(* IEC 61131-3 sources: Building-Automation/Wastewater Treatment Plant/plc, 7 files *)

(* ---- global_vars.st ---- *)
(* Wastewater Treatment Plant - Global Variables *)
VAR_GLOBAL
    (* Digital Inputs *)
    INTAKE_FLOW AT %I0.0 : BOOL;              (* Intake flow switch *)
    OUTFLOW_SENSOR AT %I0.1 : BOOL;           (* Treated water flow *)
    TANK_HIGH_LEVEL AT %I0.2 : BOOL;          (* High level switch *)
    EMERGENCY_STOP AT %I0.3 : BOOL;           (* Emergency stop *)
    SCREEN_CLOG AT %I0.4 : BOOL;              (* Screen clog detection *)
    AERATION_RUNNING AT %I0.5 : BOOL;         (* Aeration status *)
    PUMP_P101_RUNNING AT %I0.6 : BOOL;        (* Primary pump status *)
    PUMP_P102_RUNNING AT %I0.7 : BOOL;        (* Secondary pump status *)
    CHLORINE_LOW AT %I1.0 : BOOL;             (* Chlorine level low *)
    ACID_TANK_LOW AT %I1.1 : BOOL;            (* pH adjustment low *)
    GAS_ALARM AT %I1.2 : BOOL;                (* Gas detection *)
    AUTO_MODE AT %I1.3 : BOOL;                (* Auto mode selection *)
    FILTER_PRESSURE_HIGH AT %I1.4 : BOOL;     (* Filter differential *)
    UV_SYSTEM_RUNNING AT %I1.5 : BOOL;        (* UV disinfection status *)
    SLUDGE_PUMP_RUNNING AT %I1.6 : BOOL;      (* Sludge pump status *)
    MAINTENANCE_MODE AT %I1.7 : BOOL;         (* Maintenance switch *)

    (* Digital Outputs *)
    PUMP_P101_START AT %Q0.0 : BOOL;          (* Primary pump start *)
    PUMP_P102_START AT %Q0.1 : BOOL;          (* Secondary pump start *)
    MIXER_M101_START AT %Q0.2 : BOOL;         (* Primary mixer start *)
    MIXER_M102_START AT %Q0.3 : BOOL;         (* Secondary mixer start *)
    SCREEN_FORWARD AT %Q0.4 : BOOL;           (* Screen forward *)
    SCREEN_REVERSE AT %Q0.5 : BOOL;           (* Screen reverse *)
    BLOWER_START AT %Q0.6 : BOOL;             (* Aeration blower *)
    UV_SYSTEM_START AT %Q0.7 : BOOL;          (* UV system start *)
    ACID_DOSING_PUMP AT %Q1.0 : BOOL;         (* Acid dosing *)
    BASE_DOSING_PUMP AT %Q1.1 : BOOL;         (* Base dosing *)
    CHLORINE_DOSING AT %Q1.2 : BOOL;          (* Chlorine dosing *)
    SLUDGE_PUMP_START AT %Q1.3 : BOOL;        (* Sludge pump start *)
    ALARM_BEACON AT %Q1.4 : BOOL;             (* Visual alarm *)
    ALARM_HORN AT %Q1.5 : BOOL;               (* Audible alarm *)
    BACKWASH_VALVE AT %Q1.6 : BOOL;           (* Filter backwash *)
    OUTLET_VALVE AT %Q1.7 : BOOL;             (* Outlet control *)

    (* Analog Inputs *)
    INTAKE_FLOW_RATE AT %IW0 : INT;           (* Intake flow meter 0-600m³/h *)
    OUTPUT_FLOW_RATE AT %IW1 : INT;           (* Output flow meter 0-600m³/h *)
    TANK_LEVEL_1 AT %IW2 : INT;               (* Primary tank level 0-5m *)
    TANK_LEVEL_2 AT %IW3 : INT;               (* Secondary tank level 0-5m *)
    PH_VALUE AT %IW4 : INT;                   (* pH measurement 0-14 pH *)
    DISSOLVED_OXYGEN AT %IW5 : INT;           (* DO measurement 0-20mg/L *)
    TURBIDITY AT %IW6 : INT;                  (* Turbidity meter 0-1000NTU *)
    TEMPERATURE AT %IW7 : INT;                (* Process temperature 0-100°C *)
    CONDUCTIVITY AT %IW8 : INT;               (* Conductivity meter 0-5000µS/cm *)
    CHLORINE_RESIDUAL AT %IW9 : INT;          (* Chlorine analyzer 0-10mg/L *)
    POWER_CONSUMPTION AT %IW10 : INT;         (* System power 0-500kW *)
    PRESSURE_SENSOR_1 AT %IW11 : INT;         (* Process pressure 1 0-10bar *)

    (* Analog Outputs *)
    PUMP_P101_SPEED AT %QW0 : INT;            (* Primary pump VFD 0-100% *)
    PUMP_P102_SPEED AT %QW1 : INT;            (* Secondary pump VFD 0-100% *)
    BLOWER_SPEED AT %QW2 : INT;               (* Aeration blower VFD 0-100% *)
    ACID_DOSING_RATE AT %QW3 : INT;           (* Acid dosing rate 0-100% *)
    BASE_DOSING_RATE AT %QW4 : INT;           (* Base dosing rate 0-100% *)
    CHLORINE_DOSING_RATE AT %QW5 : INT;       (* Chlorine dose rate 0-100% *)
    MIXER_M101_SPEED AT %QW6 : INT;           (* Primary mixer VFD 0-100% *)
    MIXER_M102_SPEED AT %QW7 : INT;           (* Secondary mixer VFD 0-100% *)

    (* System Status Variables *)
    SystemRunning : BOOL;                     (* Overall system running status *)
    SystemFault : BOOL;                       (* System fault status *)
    MaintenanceRequired : BOOL;               (* Maintenance required indicator *)
    BatchProcessing : BOOL;                   (* Batch processing mode active *)
    StormModeActive : BOOL;                   (* Storm water handling mode *)

    (* Alarms and Warnings *)
    AlarmActive : BOOL;                       (* Any alarm active *)
    HighPHAlarm : BOOL;                       (* pH too high alarm *)
    LowPHAlarm : BOOL;                        (* pH too low alarm *)
    HighTurbidityAlarm : BOOL;                (* High turbidity alarm *)
    LowOxygenAlarm : BOOL;                    (* Low dissolved oxygen alarm *)
    ChemicalLevelWarning : BOOL;              (* Chemical level warning *)
    GasDetectionAlarm : BOOL;                 (* Hazardous gas detected *)

    (* Process Setpoints *)
    PHSetpoint : REAL := 7.0;                 (* pH setpoint (typically 6.5-8.5) *)
    DissolvedOxygenSetpoint : REAL := 5.0;    (* DO setpoint (mg/L) *)
    ChlorineDosageSetpoint : REAL := 2.5;     (* Chlorine dosage setpoint (mg/L) *)
    FlowRateSetpoint : REAL := 300.0;         (* Flow rate setpoint (m³/h) *)

    (* Process Variables (scaled) *)
    ScaledPHValue : REAL;                     (* Scaled pH value (0-14) *)
    ScaledDO : REAL;                          (* Scaled dissolved oxygen (mg/L) *)
    ScaledTurbidity : REAL;                   (* Scaled turbidity (NTU) *)
    ScaledFlowRate : REAL;                    (* Scaled flow rate (m³/h) *)
    ScaledTankLevel1 : REAL;                  (* Scaled primary tank level (m) *)
    ScaledTankLevel2 : REAL;                  (* Scaled secondary tank level (m) *)
    ScaledChlorineResidual : REAL;            (* Scaled chlorine residual (mg/L) *)

    (* Timers and Counters *)
    BackwashTimer : TON;                      (* Filter backwash timer *)
    ChemicalDosingTimer : TON;                (* Chemical dosing timer *)
    ProcessCycleTimer : TON;                  (* Process cycle timer *)
    MaintenanceCounter : CTU;                 (* Maintenance interval counter *)

    (* PID Controllers *)
    PHController : PID;                       (* pH control PID *)
    DOController : PID;                       (* Dissolved oxygen PID *)
    FlowController : PID;                     (* Flow rate PID *)
    ChlorineController : PID;                 (* Chlorine dosing PID *)

    (* Statistical Data *)
    TotalFlowToday : REAL;                    (* Daily flow totalization (m³) *)
    TotalChemicalUsage : REAL;                (* Chemical usage (L) *)
    TotalEnergyUsage : REAL;                  (* Energy usage (kWh) *)
    TreatmentEfficiency : REAL;               (* Treatment efficiency (%) *)

    (* System Parameters *)
    MAX_FLOW_RATE : REAL := 600.0;            (* Maximum flow rate (m³/h) *)
    MAX_TANK_LEVEL : REAL := 5.0;             (* Maximum tank level (m) *)
    MIN_PH : REAL := 6.0;                     (* Minimum allowable pH *)
    MAX_PH : REAL := 9.0;                     (* Maximum allowable pH *)
    MIN_DO : REAL := 2.0;                     (* Minimum dissolved oxygen (mg/L) *)
    MAX_TURBIDITY : REAL := 100.0;            (* Maximum allowable turbidity (NTU) *)
END_VAR

(* ---- aeration_controller.st ---- *)
PROGRAM aeration_controller
VAR
    DOPIDParams : PID_PARAMS;
    DOController : PID;
    DOControlOutput : REAL;
    BlowerSpeedOutput : REAL := 0.0;
    AerationCycle : INT := 0;
    AerationTimer : TON;
    AerationPauseTimer : TON;
    CycleActive : BOOL := FALSE;
    MinimumBlowerSpeed : REAL := 20.0;
    MaximumBlowerSpeed : REAL := 95.0;
    BlowerStartupSequence : BOOL := FALSE;
    BlowerStartupTimer : TON;
    BlowerStartupStage : INT := 0;
    BlowerShutdownSequence : BOOL := FALSE;
    BlowerShutdownTimer : TON;
    PreviousDO : REAL := 0.0;
    DOChangeRate : REAL := 0.0;
    DOCalculationTimer : TON;
    AnoxicCycleRequired : BOOL := FALSE;
END_VAR

(* Aeration System Controller *)
(* Manages the aeration blowers and dissolved oxygen control *)

(* Only run when system is operational *)
IF SystemRunning AND SystemState < 4 THEN

    (* Calculate DO change rate every 2 minutes *)
    DOCalculationTimer(IN := TRUE, PT := T#2M);
    IF DOCalculationTimer.Q THEN
        DOChangeRate := (ScaledDO - PreviousDO) / 120.0; (* mg/L per second *)
        PreviousDO := ScaledDO;
        DOCalculationTimer(IN := FALSE);
        DOCalculationTimer(IN := TRUE, PT := T#2M);
    END_IF

    (* Check if anoxic cycle is required for nutrient removal *)
    AnoxicCycleRequired := FALSE; (* In real system, this would be based on ammonia and nitrate measurements *)

    (* Dissolved Oxygen Control *)
    IF OperatingMode = 1 AND NOT MaintenanceRequired THEN
        (* Configure DO PID controller *)
        DOPIDParams.Kp := 10.0;   (* Proportional gain *)
        DOPIDParams.Ki := 0.1;    (* Integral gain *)
        DOPIDParams.Kd := 1.0;    (* Derivative gain *)
        DOPIDParams.Deadband := 0.1; (* Deadband to prevent oscillations *)
        DOPIDParams.MaxOutput := MaximumBlowerSpeed; (* Output range *)
        DOPIDParams.MinOutput := MinimumBlowerSpeed;

        (* Execute DO PID control *)
        DOController.Parameters := DOPIDParams;
        DOController.Setpoint := DissolvedOxygenSetpoint;
        DOController.ProcessValue := ScaledDO;
        DOController.Execute();
        DOControlOutput := DOController.Output;

        (* Aeration Control Strategy - Cycle as needed *)
        CASE AerationCycle OF
            0: (* Normal aeration phase *)
                IF NOT AnoxicCycleRequired THEN
                    (* Continuous aeration based on DO control *)
                    BlowerSpeedOutput := DOControlOutput;

                    (* Ensure the blower runs at a reasonable speed *)
                    IF BlowerSpeedOutput < MinimumBlowerSpeed THEN
                        IF ScaledDO < (DissolvedOxygenSetpoint * 1.5) THEN
                            BlowerSpeedOutput := MinimumBlowerSpeed;
                        END_IF
                    END_IF

                    (* Stay in continuous mode *)
                    CycleActive := FALSE;
                ELSE
                    (* Begin cycle operation with aeration phase *)
                    AerationTimer(IN := TRUE, PT := T#30M);
                    CycleActive := TRUE;

                    (* Run blower at calculated speed *)
                    BlowerSpeedOutput := DOControlOutput;

                    (* Move to anoxic phase after timer expires *)
                    IF AerationTimer.Q THEN
                        AerationCycle := 1;
                        AerationTimer(IN := FALSE);
                        AerationPauseTimer(IN := FALSE);
                    END_IF
                END_IF

            1: (* Anoxic phase - blower off for denitrification *)
                BlowerSpeedOutput := 0.0;
                AerationPauseTimer(IN := TRUE, PT := T#45M);

                (* Emergency override - if DO drops too low, restart aeration *)
                IF ScaledDO < (MIN_DO * 0.5) THEN
                    AerationCycle := 0;
                    AerationPauseTimer(IN := FALSE);
                END_IF

                (* Return to aeration phase after timer expires *)
                IF AerationPauseTimer.Q THEN
                    AerationCycle := 0;
                    AerationPauseTimer(IN := FALSE);
                END_IF
        END_CASE

        (* Blower Startup Sequence *)
        IF BlowerSpeedOutput > 0.0 AND NOT BLOWER_START THEN
            (* Initialize startup sequence *)
            BlowerStartupSequence := TRUE;
            BlowerShutdownSequence := FALSE;
            BlowerStartupStage := 0;
            BlowerStartupTimer(IN := FALSE);
        END_IF

        (* Blower Shutdown Sequence *)
        IF BlowerSpeedOutput = 0.0 AND BLOWER_START THEN
            (* Initialize shutdown sequence *)
            BlowerShutdownSequence := TRUE;
            BlowerStartupSequence := FALSE;
            BlowerShutdownTimer(IN := FALSE);
        END_IF

        (* Execute Blower Startup Sequence *)
        IF BlowerStartupSequence THEN
            CASE BlowerStartupStage OF
                0: (* Pre-start checks *)
                    BLOWER_START := FALSE;
                    BLOWER_SPEED := 0;
                    BlowerStartupTimer(IN := TRUE, PT := T#5S);
                    IF BlowerStartupTimer.Q THEN
                        BlowerStartupStage := 1;
                        BlowerStartupTimer(IN := FALSE);
                    END_IF

                1: (* Start motor *)
                    BLOWER_START := TRUE;
                    BLOWER_SPEED := REAL_TO_INT(MinimumBlowerSpeed * 27648.0 / 100.0);
                    BlowerStartupTimer(IN := TRUE, PT := T#10S);
                    IF BlowerStartupTimer.Q THEN
                        BlowerStartupStage := 2;
                        BlowerStartupTimer(IN := FALSE);
                    END_IF

                2: (* Ramp up to target speed *)
                    BLOWER_SPEED := REAL_TO_INT(BlowerSpeedOutput * 27648.0 / 100.0);
                    BlowerStartupSequence := FALSE;
            END_CASE
        END_IF

        (* Execute Blower Shutdown Sequence *)
        IF BlowerShutdownSequence THEN
            (* Ramp down speed first *)
            BLOWER_SPEED := REAL_TO_INT(MinimumBlowerSpeed * 27648.0 / 100.0);
            BlowerShutdownTimer(IN := TRUE, PT := T#15S);

            IF BlowerShutdownTimer.Q THEN
                (* Safe to stop motor *)
                BLOWER_START := FALSE;
                BLOWER_SPEED := 0;
                BlowerShutdownSequence := FALSE;
                BlowerShutdownTimer(IN := FALSE);
            END_IF
        END_IF

        (* Update blower speed if running and not in startup/shutdown sequence *)
        IF BLOWER_START AND NOT BlowerStartupSequence AND NOT BlowerShutdownSequence THEN
            (* Smooth out rapid DO changes to prevent blower hunting *)
            IF ABS(DOChangeRate) > 0.005 THEN
                (* DO changing quickly - apply more gradual change to blower speed *)
                BlowerSpeedOutput := 0.7 * BlowerSpeedOutput + 0.3 * REAL_TO_INT(BLOWER_SPEED) * 100.0 / 27648.0;
            END_IF

            (* Apply control output to blower *)
            BLOWER_SPEED := REAL_TO_INT(BlowerSpeedOutput * 27648.0 / 100.0);
        END_IF

    ELSIF OperatingMode = 2 THEN
        (* Storm mode - maximum aeration capacity *)
        BLOWER_START := TRUE;
        BLOWER_SPEED := REAL_TO_INT(MaximumBlowerSpeed * 27648.0 / 100.0);

    ELSIF OperatingMode = 3 THEN
        (* Maintenance mode - manually controlled from HMI *)
        (* Keep current state - will be controlled by direct PLC writes *)
    ELSE
        (* System stopped or fault - ensure blower is off *)
        BLOWER_START := FALSE;
        BLOWER_SPEED := 0;
    END_IF

END_IF

END_PROGRAM

(* ---- dosing_controller.st ---- *)
PROGRAM dosing_controller
VAR
    PHPIDParams : PID_PARAMS;
    ChlorinePIDParams : PID_PARAMS;
    PHController : PID;
    ChlorineController : PID;
    PHControlOutput : REAL;
    ChlorineControlOutput : REAL;
    AcidDosingActive : BOOL := FALSE;
    BaseDosingActive : BOOL := FALSE;
    ChlorineDosingActive : BOOL := FALSE;
    ChemicalPulseTimer : TON;
    ChemicalPulseActive : BOOL := FALSE;
    DosingDisabled : BOOL := FALSE;
    DosingRate : REAL := 0.0;
    ChlorineDosingRate : REAL := 0.0;
    UrgentPHCorrection : BOOL := FALSE;
    PreviousPHValue : REAL := 7.0;
    PHChangeRate : REAL := 0.0;
    PHCalculationTimer : TON;
END_VAR

(* Chemical Dosing Controller *)
(* Manages chemical dosing for pH control and disinfection *)

(* Only run when system is operational *)
IF SystemRunning AND SystemState < 4 THEN

    (* Calculate pH change rate every minute *)
    PHCalculationTimer(IN := TRUE, PT := T#1M);
    IF PHCalculationTimer.Q THEN
        PHChangeRate := (ScaledPHValue - PreviousPHValue) / 60.0; (* pH units per second *)
        PreviousPHValue := ScaledPHValue;
        PHCalculationTimer(IN := FALSE);
        PHCalculationTimer(IN := TRUE, PT := T#1M);
    END_IF

    (* Check if urgent pH correction is needed *)
    UrgentPHCorrection := (ScaledPHValue < MIN_PH - 0.5) OR (ScaledPHValue > MAX_PH + 0.5);

    (* Disable dosing during certain conditions *)
    DosingDisabled := (SystemState = 4) OR TANK_HIGH_LEVEL OR MaintenanceRequired OR
                     (ScaledTankLevel1 < 0.1) OR (ScaledFlowRate < 10.0);

    (* pH Control *)
    IF NOT DosingDisabled AND OperatingMode = 1 THEN
        (* Configure pH PID controller *)
        PHPIDParams.Kp := 5.0;   (* Proportional gain *)
        PHPIDParams.Ki := 0.2;   (* Integral gain *)
        PHPIDParams.Kd := 1.0;   (* Derivative gain *)
        PHPIDParams.Deadband := 0.1; (* Deadband to prevent oscillations *)
        PHPIDParams.MaxOutput := 100.0; (* 0-100% output range *)
        PHPIDParams.MinOutput := 0.0;

        (* Execute pH PID control *)
        PHController.Parameters := PHPIDParams;
        PHController.Setpoint := PHSetpoint;
        PHController.ProcessValue := ScaledPHValue;
        PHController.Execute();
        PHControlOutput := PHController.Output;

        (* Determine if acid or base dosing is needed *)
        IF ScaledPHValue > (PHSetpoint + 0.2) THEN
            (* pH too high - need acid *)
            AcidDosingActive := TRUE;
            BaseDosingActive := FALSE;

            (* Calculate acid dosing rate, proportional to deviation *)
            DosingRate := PHControlOutput;

            (* Apply limits and safety checks *)
            IF ACID_TANK_LOW THEN
                DosingRate := DosingRate * 0.5; (* Reduce dosing when supply low *)
            END_IF

            (* Convert to PLC output format *)
            ACID_DOSING_RATE := REAL_TO_INT(DosingRate * 27648.0 / 100.0);
            BASE_DOSING_RATE := 0;

            (* Control dosing pump *)
            ACID_DOSING_PUMP := (DosingRate > 5.0);
            BASE_DOSING_PUMP := FALSE;

        ELSIF ScaledPHValue < (PHSetpoint - 0.2) THEN
            (* pH too low - need base *)
            AcidDosingActive := FALSE;
            BaseDosingActive := TRUE;

            (* Calculate base dosing rate, proportional to deviation *)
            DosingRate := PHControlOutput;

            (* Apply limits and safety checks *)
            IF ABS(PHChangeRate) > 0.01 THEN
                (* pH changing quickly - reduce dosing to prevent overshooting *)
                DosingRate := DosingRate * 0.7;
            END_IF

            (* Convert to PLC output format *)
            ACID_DOSING_RATE := 0;
            BASE_DOSING_RATE := REAL_TO_INT(DosingRate * 27648.0 / 100.0);

            (* Control dosing pump *)
            ACID_DOSING_PUMP := FALSE;
            BASE_DOSING_PUMP := (DosingRate > 5.0);

        ELSE
            (* pH within acceptable range - no dosing needed *)
            AcidDosingActive := FALSE;
            BaseDosingActive := FALSE;
            ACID_DOSING_PUMP := FALSE;
            BASE_DOSING_PUMP := FALSE;
            ACID_DOSING_RATE := 0;
            BASE_DOSING_RATE := 0;
        END_IF

        (* Disinfection Control - Chlorine Dosing *)
        IF OUTLET_VALVE AND ScaledFlowRate > 20.0 THEN
            (* Configure chlorine PID controller *)
            ChlorinePIDParams.Kp := 3.0;   (* Proportional gain *)
            ChlorinePIDParams.Ki := 0.1;   (* Integral gain *)
            ChlorinePIDParams.Kd := 0.5;   (* Derivative gain *)
            ChlorinePIDParams.Deadband := 0.05; (* Deadband to prevent oscillations *)
            ChlorinePIDParams.MaxOutput := 100.0; (* 0-100% output range *)
            ChlorinePIDParams.MinOutput := 0.0;

            (* Execute chlorine PID control *)
            ChlorineController.Parameters := ChlorinePIDParams;
            ChlorineController.Setpoint := ChlorineDosageSetpoint;
            ChlorineController.ProcessValue := ScaledChlorineResidual;
            ChlorineController.Execute();
            ChlorineControlOutput := ChlorineController.Output;

            (* Apply chlorine dosing *)
            ChlorineDosingActive := TRUE;

            (* Calculate dosing rate with flow-based adjustment *)
            ChlorineDosingRate := ChlorineControlOutput * (ScaledFlowRate / FlowRateSetpoint);

            (* Apply limits and safety checks *)
            IF CHLORINE_LOW THEN
                ChlorineDosingRate := ChlorineDosingRate * 0.5; (* Reduce when supply low *)
            END_IF

            (* Convert to PLC output format *)
            CHLORINE_DOSING_RATE := REAL_TO_INT(ChlorineDosingRate * 27648.0 / 100.0);

            (* Control dosing pump *)
            CHLORINE_DOSING := (ChlorineDosingRate > 5.0);

            (* Track chemical usage *)
            IF CHLORINE_DOSING THEN
                TotalChemicalUsage := TotalChemicalUsage + (ChlorineDosingRate * 0.001); (* L per cycle *)
            END_IF

        ELSE
            (* No outlet flow - stop chlorine dosing *)
            ChlorineDosingActive := FALSE;
            CHLORINE_DOSING := FALSE;
            CHLORINE_DOSING_RATE := 0;
        END_IF

    ELSE
        (* System in fault or manual mode - disable all chemical dosing *)
        AcidDosingActive := FALSE;
        BaseDosingActive := FALSE;
        ChlorineDosingActive := FALSE;
        ACID_DOSING_PUMP := FALSE;
        BASE_DOSING_PUMP := FALSE;
        CHLORINE_DOSING := FALSE;
        ACID_DOSING_RATE := 0;
        BASE_DOSING_RATE := 0;
        CHLORINE_DOSING_RATE := 0;
    END_IF

    (* Pulse-based dosing for more precise chemical control *)
    IF (AcidDosingActive OR BaseDosingActive OR ChlorineDosingActive) AND DosingRate > 0.0 THEN
        ChemicalPulseTimer(IN := TRUE, PT := T#10S);
        IF ChemicalPulseTimer.Q THEN
            ChemicalPulseTimer(IN := FALSE);
            ChemicalPulseActive := NOT ChemicalPulseActive;

            (* Modify dosing pattern based on pulse state *)
            IF ChemicalPulseActive THEN
                IF AcidDosingActive THEN
                    ACID_DOSING_PUMP := TRUE;
                END_IF
                IF BaseDosingActive THEN
                    BASE_DOSING_PUMP := TRUE;
                END_IF
                IF ChlorineDosingActive THEN
                    CHLORINE_DOSING := TRUE;
                END_IF
            ELSE
                (* Keep pumps running for high demand, otherwise pulse them *)
                IF AcidDosingActive AND DosingRate < 30.0 AND NOT UrgentPHCorrection THEN
                    ACID_DOSING_PUMP := FALSE;
                END_IF
                IF BaseDosingActive AND DosingRate < 30.0 AND NOT UrgentPHCorrection THEN
                    BASE_DOSING_PUMP := FALSE;
                END_IF
                IF ChlorineDosingActive AND ChlorineDosingRate < 20.0 THEN
                    CHLORINE_DOSING := FALSE;
                END_IF
            END_IF
        END_IF
    ELSE
        ChemicalPulseTimer(IN := FALSE);
    END_IF

END_IF

END_PROGRAM

(* ---- intake_controller.st ---- *)
PROGRAM intake_controller
VAR
    ScreenCleaningTimer : TON;
    ScreenCleaningActive : BOOL := FALSE;
    ScreenCleaningCycle : INT := 0;
    IntakeValvePosition : INT := 0;
    FlowSetpoint : REAL := 300.0; (* Default flow setpoint *)
    FlowPIDParams : PID_PARAMS;
    ScreeningActive : BOOL := FALSE;
    FlowControl : PID;
    FlowControlOutput : REAL;
    ManualOverrideActive : BOOL := FALSE;
    ScreenClogDetected : BOOL := FALSE;
    PreviousScreenClog : BOOL := FALSE;
END_VAR

(* Intake Process Controller *)
(* Manages the initial wastewater intake, screening, and flow control *)

(* Only run when system is operational *)
IF SystemRunning AND SystemState < 4 THEN

    (* Screen Clog Detection *)
    ScreenClogDetected := SCREEN_CLOG;
    IF ScreenClogDetected AND NOT PreviousScreenClog THEN
        (* New clog detected - start cleaning cycle *)
        ScreenCleaningTimer(IN := FALSE);
        ScreenCleaningActive := TRUE;
        ScreenCleaningCycle := 0;
    END_IF
    PreviousScreenClog := ScreenClogDetected;

    (* Screening System Control *)
    IF ScreenCleaningActive THEN
        (* Screen Cleaning Sequence *)
        CASE ScreenCleaningCycle OF
            0: (* Forward motion *)
                SCREEN_FORWARD := TRUE;
                SCREEN_REVERSE := FALSE;
                ScreenCleaningTimer(IN := TRUE, PT := T#30S);
                IF ScreenCleaningTimer.Q THEN
                    ScreenCleaningTimer(IN := FALSE);
                    ScreenCleaningCycle := 1;
                END_IF

            1: (* Stop briefly *)
                SCREEN_FORWARD := FALSE;
                SCREEN_REVERSE := FALSE;
                ScreenCleaningTimer(IN := TRUE, PT := T#5S);
                IF ScreenCleaningTimer.Q THEN
                    ScreenCleaningTimer(IN := FALSE);
                    ScreenCleaningCycle := 2;
                END_IF

            2: (* Reverse motion *)
                SCREEN_FORWARD := FALSE;
                SCREEN_REVERSE := TRUE;
                ScreenCleaningTimer(IN := TRUE, PT := T#20S);
                IF ScreenCleaningTimer.Q THEN
                    ScreenCleaningTimer(IN := FALSE);
                    ScreenCleaningCycle := 3;
                END_IF

            3: (* Complete cycle *)
                SCREEN_FORWARD := FALSE;
                SCREEN_REVERSE := FALSE;
                ScreenCleaningActive := FALSE;
        END_CASE
    ELSIF OperatingMode = 1 THEN
        (* Normal screening operation *)
        (* Run screen periodically with timer based on flow rate *)
        IF ScaledFlowRate > 100.0 THEN
            SCREEN_FORWARD := TRUE;
            SCREEN_REVERSE := FALSE;
            ScreeningActive := TRUE;
        ELSE
            IF ScreeningActive THEN
                ScreenCleaningTimer(IN := TRUE, PT := T#60S);
                IF ScreenCleaningTimer.Q THEN
                    SCREEN_FORWARD := FALSE;
                    SCREEN_REVERSE := FALSE;
                    ScreeningActive := FALSE;
                    ScreenCleaningTimer(IN := FALSE);
                END_IF
            END_IF
        END_IF
    ELSE
        (* Maintenance mode or storm mode - manual control from HMI *)
        (* Keep current state - will be controlled directly by Q variables *)
    END_IF

    (* Flow Control *)
    IF OperatingMode = 1 AND NOT ManualOverrideActive THEN
        (* Auto mode flow control *)
        (* Set flow rate based on current system capacity *)
        IF SystemState = 1 THEN
            (* Normal operation *)
            FlowSetpoint := FlowRateSetpoint; (* From global setpoint *)
        ELSIF SystemState = 2 THEN
            (* Warning state - reduce flow *)
            FlowSetpoint := FlowRateSetpoint * 0.8;
        ELSIF SystemState = 3 THEN
            (* Alarm state - further reduce flow *)
            FlowSetpoint := FlowRateSetpoint * 0.5;
        END_IF

        (* Scale back if tanks are getting too full *)
        IF ScaledTankLevel1 > (MAX_TANK_LEVEL * 0.9) THEN
            FlowSetpoint := FlowSetpoint * 0.7;
        END_IF

        (* Storm mode override *)
        IF OperatingMode = 2 THEN
            FlowSetpoint := MAX_FLOW_RATE * 0.9; (* Near maximum capacity *)
        END_IF

        (* Configure PID controller *)
        FlowPIDParams.Kp := 2.0;   (* Proportional gain *)
        FlowPIDParams.Ki := 0.1;   (* Integral gain *)
        FlowPIDParams.Kd := 0.05;  (* Derivative gain *)
        FlowPIDParams.Deadband := 5.0; (* Deadband to prevent oscillations *)
        FlowPIDParams.MaxOutput := 100.0; (* 0-100% output range *)
        FlowPIDParams.MinOutput := 0.0;

        (* Execute PID control *)
        FlowControl.Parameters := FlowPIDParams;
        FlowControl.Setpoint := FlowSetpoint;
        FlowControl.ProcessValue := ScaledFlowRate;
        FlowControl.Execute();
        FlowControlOutput := FlowControl.Output;

        (* Apply control output to pump *)
        IF INTAKE_FLOW OR ScaledFlowRate < 10.0 THEN
            PUMP_P101_START := TRUE;
            PUMP_P101_SPEED := REAL_TO_INT(FlowControlOutput * 27648.0 / 100.0);
        ELSE
            (* No flow detected at input - stop pump *)
            PUMP_P101_START := FALSE;
            PUMP_P101_SPEED := 0;
        END_IF
    ELSIF OperatingMode = 3 THEN
        (* Maintenance mode - commands from HMI *)
        (* Keep last state - will be controlled by direct PLC writes *)
    END_IF

    (* Valve control based on tank levels *)
    IF ScaledTankLevel1 > MAX_TANK_LEVEL * 0.95 THEN
        (* Close inlet valve to prevent overflow *)
        IntakeValvePosition := 0;
    ELSIF ScaledFlowRate < 20.0 AND PUMP_P101_START THEN
        (* Possible blockage or dry run - reduce valve opening *)
        IntakeValvePosition := 3000; (* ~10% *)
    ELSE
        (* Normal operation - valve position follows flow demand *)
        IntakeValvePosition := 8000 + REAL_TO_INT(FlowControlOutput * 19000.0 / 100.0);
    END_IF
END_IF

END_PROGRAM

(* ---- main.st ---- *)
PROGRAM main
VAR
    FirstScan : BOOL := TRUE;
    OperatingMode : INT := 0; (* 0: Stopped, 1: Auto, 2: Storm, 3: Maintenance *)
    SystemState : INT := 0;   (* 0: Init, 1: Running, 2: Warning, 3: Alarm, 4: Emergency *)
    StartupSequenceComplete : BOOL := FALSE;
    SystemInitTimer : TON;
    HeartbeatTimer : TON;
    HeartbeatPulse : BOOL := FALSE;
    PulseTimer : TON;
END_VAR

(* Main control program for Wastewater Treatment Plant *)
(* This program coordinates all subsystems and manages overall plant operations *)

(* System Initialization *)
IF FirstScan THEN
    SystemInitTimer(IN := TRUE, PT := T#10S);
    HeartbeatTimer(IN := TRUE, PT := T#1S);
    PulseTimer(IN := TRUE, PT := T#500MS);
    FirstScan := FALSE;
    SystemRunning := FALSE;
    SystemFault := FALSE;
    AlarmActive := FALSE;

    (* Reset all outputs to safe state *)
    PUMP_P101_START := FALSE;
    PUMP_P102_START := FALSE;
    MIXER_M101_START := FALSE;
    MIXER_M102_START := FALSE;
    SCREEN_FORWARD := FALSE;
    SCREEN_REVERSE := FALSE;
    BLOWER_START := FALSE;
    UV_SYSTEM_START := FALSE;
    ACID_DOSING_PUMP := FALSE;
    BASE_DOSING_PUMP := FALSE;
    CHLORINE_DOSING := FALSE;
    SLUDGE_PUMP_START := FALSE;
    ALARM_BEACON := FALSE;
    ALARM_HORN := FALSE;
    BACKWASH_VALVE := FALSE;
    OUTLET_VALVE := FALSE;

    (* Initialize analog outputs *)
    PUMP_P101_SPEED := 0;
    PUMP_P102_SPEED := 0;
    BLOWER_SPEED := 0;
    ACID_DOSING_RATE := 0;
    BASE_DOSING_RATE := 0;
    CHLORINE_DOSING_RATE := 0;
    MIXER_M101_SPEED := 0;
    MIXER_M102_SPEED := 0;
END_IF

(* Determine System State Based on Inputs *)
IF EMERGENCY_STOP THEN
    SystemState := 4; (* Emergency *)
ELSIF GAS_ALARM OR HighPHAlarm OR LowPHAlarm OR HighTurbidityAlarm OR LowOxygenAlarm THEN
    SystemState := 3; (* Alarm *)
ELSIF ChemicalLevelWarning OR SCREEN_CLOG OR FILTER_PRESSURE_HIGH THEN
    SystemState := 2; (* Warning *)
ELSIF StartupSequenceComplete THEN
    SystemState := 1; (* Running *)
ELSE
    SystemState := 0; (* Initializing *)
END_IF

(* System Initialization Sequence *)
IF SystemInitTimer.Q AND NOT StartupSequenceComplete THEN
    (* Initialization complete, system ready to run *)
    StartupSequenceComplete := TRUE;
END_IF

(* Determine Operating Mode *)
IF MAINTENANCE_MODE THEN
    OperatingMode := 3; (* Maintenance *)
ELSIF StormModeActive THEN
    OperatingMode := 2; (* Storm *)
ELSIF AUTO_MODE AND StartupSequenceComplete THEN
    OperatingMode := 1; (* Automatic *)
ELSE
    OperatingMode := 0; (* Stopped *)
END_IF

(* System Heartbeat *)
HeartbeatTimer();
IF HeartbeatTimer.Q THEN
    HeartbeatPulse := NOT HeartbeatPulse;
    HeartbeatTimer(IN := TRUE, PT := T#1S);
END_IF

(* Fast Pulse for Controllers *)
PulseTimer();
IF PulseTimer.Q THEN
    PulseTimer(IN := TRUE, PT := T#500MS);
END_IF

(* Process measurements and scale analog inputs *)
ScaledFlowRate := INT_TO_REAL(INTAKE_FLOW_RATE) * MAX_FLOW_RATE / 27648.0;
ScaledTankLevel1 := INT_TO_REAL(TANK_LEVEL_1) * MAX_TANK_LEVEL / 27648.0;
ScaledTankLevel2 := INT_TO_REAL(TANK_LEVEL_2) * MAX_TANK_LEVEL / 27648.0;
ScaledPHValue := 14.0 * INT_TO_REAL(PH_VALUE) / 27648.0;
ScaledDO := 20.0 * INT_TO_REAL(DISSOLVED_OXYGEN) / 27648.0;
ScaledTurbidity := 1000.0 * INT_TO_REAL(TURBIDITY) / 27648.0;
ScaledChlorineResidual := 10.0 * INT_TO_REAL(CHLORINE_RESIDUAL) / 27648.0;

(* Alarm Evaluation *)
HighPHAlarm := ScaledPHValue > MAX_PH;
LowPHAlarm := ScaledPHValue < MIN_PH AND ScaledPHValue > 0.5; (* Ignore if near zero - likely a sensor fault *)
LowOxygenAlarm := ScaledDO < MIN_DO AND BatchProcessing;
HighTurbidityAlarm := ScaledTurbidity > MAX_TURBIDITY;
ChemicalLevelWarning := CHLORINE_LOW OR ACID_TANK_LOW;
GasDetectionAlarm := GAS_ALARM;
AlarmActive := HighPHAlarm OR LowPHAlarm OR HighTurbidityAlarm OR LowOxygenAlarm OR GasDetectionAlarm;

(* Alarm Indicators *)
ALARM_BEACON := AlarmActive OR SystemState = 4; (* On for Alarms & Emergency *)
ALARM_HORN := SystemState = 4; (* Horn only for Emergency *)

(* System Running Status *)
SystemRunning := (OperatingMode > 0) AND (SystemState < 4);
MaintenanceRequired := (OperatingMode = 3) OR SCREEN_CLOG OR FILTER_PRESSURE_HIGH;

(* Call Subsystem Controllers *)
(* Each controller manages its specific process area *)
intake_controller();
treatment_controller();
dosing_controller();
aeration_controller();
monitoring_controller();

(* Safety Interlocks Override - Emergency Stop *)
IF SystemState = 4 THEN
    (* Emergency Stop - Shutdown all processes *)
    PUMP_P101_START := FALSE;
    PUMP_P102_START := FALSE;
    MIXER_M101_START := FALSE;
    MIXER_M102_START := FALSE;
    BLOWER_START := FALSE;
    ACID_DOSING_PUMP := FALSE;
    BASE_DOSING_PUMP := FALSE;
    CHLORINE_DOSING := FALSE;
    SLUDGE_PUMP_START := FALSE;

    (* Set all analog outputs to safe state *)
    PUMP_P101_SPEED := 0;
    PUMP_P102_SPEED := 0;
    BLOWER_SPEED := 0;
    ACID_DOSING_RATE := 0;
    BASE_DOSING_RATE := 0;
    CHLORINE_DOSING_RATE := 0;
    MIXER_M101_SPEED := 0;
    MIXER_M102_SPEED := 0;

    (* Ensure outlet valve is closed *)
    OUTLET_VALVE := FALSE;
END_IF

(* Daily totalization calculation *)
IF SystemRunning THEN
    TotalFlowToday := TotalFlowToday + (ScaledFlowRate / 3600.0); (* m³/hr to m³/second *)
    TotalEnergyUsage := TotalEnergyUsage + (INT_TO_REAL(POWER_CONSUMPTION) * 500.0 / 27648.0 / 3600.0); (* kW to kWh *)
END_IF

(* Treatment Efficiency Calculation - simplified approximation *)
IF ScaledFlowRate > 10.0 AND ScaledTurbidity < MAX_TURBIDITY THEN
    TreatmentEfficiency := 100.0 * (1.0 - ScaledTurbidity / 1000.0);
END_IF

END_PROGRAM

(* ---- monitoring_controller.st ---- *)
PROGRAM monitoring_controller
VAR
    MonitoringCycleTimer : TON;
    DataLogTimer : TON;
    SampleCollectionTimer : TON;
    SampleInterval : TIME := T#4H;
    LastSampleTime : TIME;
    SampleNeeded : BOOL := FALSE;
    ComplianceCheckTimer : TON;
    ComplianceStatus : BOOL := TRUE;
    OutOfSpecCount : INT := 0;
    AlarmHistoryIndex : INT := 0;
    AlarmHistoryTime : ARRAY[0..9] OF TIME;
    AlarmHistoryCode : ARRAY[0..9] OF INT;
    LimitsExceeded : BOOL := FALSE;
    WaterQualityStatus : INT := 0; (* 0=Good, 1=Marginal, 2=Poor *)
    FirstScan : BOOL := TRUE;
    ParameterCheckCycle : INT := 0;
END_VAR

(* Monitoring and Reporting Controller *)
(* Handles monitoring, data logging, and compliance reporting *)

(* Initialize data structures on first scan *)
IF FirstScan THEN
    ComplianceStatus := TRUE;
    OutOfSpecCount := 0;
    ParameterCheckCycle := 0;
    FirstScan := FALSE;
END_IF

(* Run monitoring even when system is not in automatic mode *)
(* This ensures critical parameters are always monitored *)

(* Cyclic monitoring of parameters *)
MonitoringCycleTimer(IN := TRUE, PT := T#10S);
IF MonitoringCycleTimer.Q THEN
    (* Reset timer for next cycle *)
    MonitoringCycleTimer(IN := FALSE);
    MonitoringCycleTimer(IN := TRUE, PT := T#10S);

    (* Cycle through parameter checks to distribute processing *)
    CASE ParameterCheckCycle OF
        0: (* pH monitoring *)
            (* Check pH is within limits *)
            IF ScaledPHValue < MIN_PH OR ScaledPHValue > MAX_PH THEN
                IF NOT (HighPHAlarm OR LowPHAlarm) THEN
                    (* New pH alarm - log it *)
                    LogAlarm(10); (* Code 10 = pH out of range *)
                END_IF
            END_IF
            ParameterCheckCycle := 1;

        1: (* Dissolved oxygen monitoring *)
            (* Check DO level *)
            IF ScaledDO < MIN_DO AND BatchProcessing THEN
                IF NOT LowOxygenAlarm THEN
                    (* New DO alarm - log it *)
                    LogAlarm(20); (* Code 20 = Low oxygen *)
                END_IF
            END_IF
            ParameterCheckCycle := 2;

        2: (* Turbidity monitoring *)
            (* Check turbidity *)
            IF ScaledTurbidity > MAX_TURBIDITY THEN
                IF NOT HighTurbidityAlarm THEN
                    (* New turbidity alarm - log it *)
                    LogAlarm(30); (* Code 30 = High turbidity *)
                END_IF

                (* Adjust water quality status *)
                WaterQualityStatus := 2; (* Poor *)
            ELSIF ScaledTurbidity > (MAX_TURBIDITY * 0.7) THEN
                (* Marginal water quality *)
                WaterQualityStatus := 1; (* Marginal *)
            ELSE
                (* Good water quality *)
                WaterQualityStatus := 0; (* Good *)
            END_IF
            ParameterCheckCycle := 3;

        3: (* Gas detection *)
            IF GAS_ALARM AND NOT GasDetectionAlarm THEN
                (* New gas alarm - log it *)
                LogAlarm(40); (* Code 40 = Dangerous gas detected *)
            END_IF
            ParameterCheckCycle := 4;

        4: (* Flow monitoring *)
            (* Check for abnormal flow conditions *)
            IF PUMP_P101_RUNNING AND ScaledFlowRate < 10.0 THEN
                (* Pump running but no flow - potential blockage *)
                LogAlarm(50); (* Code 50 = Flow anomaly *)
            END_IF
            ParameterCheckCycle := 5;

        5: (* System status *)
            (* Check overall system status *)
            IF SystemState = 3 THEN
                (* System in alarm state *)
                ComplianceStatus := FALSE;
                OutOfSpecCount := OutOfSpecCount + 1;
            ELSIF SystemState = 1 AND OutOfSpecCount > 0 THEN
                (* System back to normal - decrement counter *)
                OutOfSpecCount := OutOfSpecCount - 1;
                IF OutOfSpecCount = 0 THEN
                    ComplianceStatus := TRUE;
                END_IF
            END_IF
            ParameterCheckCycle := 0; (* Restart cycle *)
    END_CASE
END_IF

(* Data Logging Functionality *)
DataLogTimer(IN := TRUE, PT := T#15M);
IF DataLogTimer.Q THEN
    (* Time to log process data *)
    DataLogTimer(IN := FALSE);
    DataLogTimer(IN := TRUE, PT := T#15M);

    (* Log key process parameters - these would typically be stored
       in a database or data historian. Here we just set a flag. *)
    LogProcessData();
END_IF

(* Sample Collection Scheduling *)
SampleCollectionTimer(IN := TRUE, PT := SampleInterval);
IF SampleCollectionTimer.Q THEN
    (* Time for routine sample *)
    SampleNeeded := TRUE;
    LastSampleTime := 0; (* Would be current time in real system *)
    SampleCollectionTimer(IN := FALSE);
    SampleCollectionTimer(IN := TRUE, PT := SampleInterval);
END_IF

(* Compliance Checking *)
ComplianceCheckTimer(IN := TRUE, PT := T#1H);
IF ComplianceCheckTimer.Q THEN
    (* Hourly compliance check *)
    ComplianceCheckTimer(IN := FALSE);
    ComplianceCheckTimer(IN := TRUE, PT := T#1H);

    (* Check discharge parameters against regulatory limits *)
    IF OUTLET_VALVE AND (
       ScaledTurbidity > MAX_TURBIDITY OR
       ScaledPHValue < MIN_PH OR
       ScaledPHValue > MAX_PH OR
       ScaledChlorineResidual > 10.0) THEN
        (* Parameters outside regulatory limits *)
        LimitsExceeded := TRUE;

        (* Log compliance issue *)
        LogAlarm(100); (* Code 100 = Compliance violation *)

        (* In a real system, this would trigger automated reporting
           to operators and potentially regulatory agencies *)
    ELSE
        LimitsExceeded := FALSE;
    END_IF
END_IF

(* Maintenance Requirements Check *)
(* Based on runtime or specific conditions *)
MaintenanceCounter();
IF MaintenanceCounter.CV > 720 THEN (* 720 hours = 30 days *)
    (* Monthly maintenance check *)
    MaintenanceRequired := TRUE;

    (* This would typically trigger work orders or maintenance alarms *)
END_IF

(* Performance Metrics Calculation *)
(* Calculate efficiency metrics based on inlet and outlet measurements *)
IF ScaledFlowRate > 10.0 AND OUTPUT_FLOW_RATE > 0 THEN
    (* Basic efficiency calculation based on turbidity reduction *)
    (* In a real system this would include multiple parameters *)
    TreatmentEfficiency := 100.0 * (1.0 - (ScaledTurbidity / 1000.0));
END_IF

(* Define the alarm logging function *)
FUNCTION LogAlarm : VOID
VAR_INPUT
    AlarmCode : INT;
END_VAR
    (* Store alarm in history array *)
    AlarmHistoryCode[AlarmHistoryIndex] := AlarmCode;
    (* In a real system, we would store the current time *)
    AlarmHistoryIndex := (AlarmHistoryIndex + 1) MOD 10;
END_FUNCTION

(* Define the data logging function *)
FUNCTION LogProcessData : VOID
    (* In a real system, this would write to a database or data historian *)
    (* For this example, we're just creating a placeholder function *)
END_FUNCTION

END_PROGRAM

(* ---- treatment_controller.st ---- *)
PROGRAM treatment_controller
VAR
    MixerControlTimer : TON;
    MixerPulseActive : BOOL := FALSE;
    SettlingPhaseActive : BOOL := FALSE;
    SettlingTimer : TON;
    TankTransferActive : BOOL := FALSE;
    TransferTimer : TON;
    PrimaryTreatmentCycle : INT := 0;
    SecondaryValvePosition : INT := 0;
    MixingIntensity : REAL := 70.0;
    PreviousTankLevel1 : REAL := 0.0;
    TankLevelDelta : REAL := 0.0;
    TankLevelRateOfChange : REAL := 0.0;
    RateCalculationTimer : TON;
    FilterOperationTimer : TON;
    FilterBackwashNeeded : BOOL := FALSE;
END_VAR

(* Treatment Process Controller *)
(* Manages the primary and secondary treatment processes *)

(* Only run when system is operational *)
IF SystemRunning AND SystemState < 4 THEN

    (* Calculate tank level rate of change every 5 minutes *)
    RateCalculationTimer(IN := TRUE, PT := T#5M);
    IF RateCalculationTimer.Q THEN
        TankLevelDelta := ScaledTankLevel1 - PreviousTankLevel1;
        TankLevelRateOfChange := TankLevelDelta / 300.0; (* m per second *)
        PreviousTankLevel1 := ScaledTankLevel1;
        RateCalculationTimer(IN := FALSE);
        RateCalculationTimer(IN := TRUE, PT := T#5M);
    END_IF

    (* Primary Treatment Processes *)
    CASE PrimaryTreatmentCycle OF
        0: (* Filling phase - already handled by intake controller *)
            IF ScaledTankLevel1 >= (MAX_TANK_LEVEL * 0.6) THEN
                PrimaryTreatmentCycle := 1;
                MixerControlTimer(IN := FALSE);
            END_IF

        1: (* Mixing phase *)
            (* Start mixer for primary tank *)
            MIXER_M101_START := TRUE;

            (* Apply variable mixing intensity based on tank level *)
            MixingIntensity := 50.0 + (ScaledTankLevel1 / MAX_TANK_LEVEL) * 50.0;
            MIXER_M101_SPEED := REAL_TO_INT(MixingIntensity * 27648.0 / 100.0);

            (* Run mixing for determined time *)
            MixerControlTimer(IN := TRUE, PT := T#20M);
            IF MixerControlTimer.Q THEN
                PrimaryTreatmentCycle := 2;
                MixerControlTimer(IN := FALSE);
                SettlingTimer(IN := FALSE);
            END_IF

        2: (* Settling phase *)
            (* Stop mixer to allow settling *)
            MIXER_M101_START := FALSE;
            MIXER_M101_SPEED := 0;
            SettlingPhaseActive := TRUE;

            (* Allow suspended solids to settle *)
            SettlingTimer(IN := TRUE, PT := T#45M);
            IF SettlingTimer.Q THEN
                PrimaryTreatmentCycle := 3;
                SettlingTimer(IN := FALSE);
                TransferTimer(IN := FALSE);
            END_IF

        3: (* Transfer to secondary treatment *)
            (* Activate transfer pump *)
            PUMP_P102_START := TRUE;
            PUMP_P102_SPEED := 13824; (* 50% speed *)
            TankTransferActive := TRUE;

            (* Transfer for specified time or until level drops *)
            TransferTimer(IN := TRUE, PT := T#30M);
            IF TransferTimer.Q OR ScaledTankLevel1 < (MAX_TANK_LEVEL * 0.15) THEN
                PrimaryTreatmentCycle := 0;
                PUMP_P102_START := FALSE;
                PUMP_P102_SPEED := 0;
                TransferTimer(IN := FALSE);
                TankTransferActive := FALSE;
            END_IF
    END_CASE

    (* Secondary Treatment Tank Control *)
    IF ScaledTankLevel2 > (MAX_TANK_LEVEL * 0.3) THEN
        (* Start secondary mixing when tank has sufficient level *)
        MIXER_M102_START := TRUE;
        MIXER_M102_SPEED := REAL_TO_INT(60.0 * 27648.0 / 100.0); (* 60% speed *)
    ELSE
        (* Tank too empty for effective mixing *)
        MIXER_M102_START := FALSE;
        MIXER_M102_SPEED := 0;
    END_IF

    (* Control outlet valve position based on treatment status *)
    IF ScaledTankLevel2 > (MAX_TANK_LEVEL * 0.5) AND
       ScaledPHValue >= MIN_PH AND ScaledPHValue <= MAX_PH AND
       ScaledTurbidity < MAX_TURBIDITY * 0.8 THEN
        (* Conditions good for discharge *)
        OUTLET_VALVE := TRUE;
    ELSE
        (* Close outlet if conditions not suitable *)
        OUTLET_VALVE := FALSE;
    END_IF

    (* Filter Operation Control *)
    IF NOT FILTER_PRESSURE_HIGH THEN
        (* Normal filter operation *)
        FilterOperationTimer(IN := TRUE, PT := T#8H);
        IF FilterOperationTimer.Q THEN
            (* Time for scheduled backwash *)
            FilterBackwashNeeded := TRUE;
            FilterOperationTimer(IN := FALSE);
        END_IF
    ELSE
        (* High pressure difference - needs immediate backwash *)
        FilterBackwashNeeded := TRUE;
    END_IF

    (* Filter Backwash Sequence *)
    IF FilterBackwashNeeded THEN
        (* Close outlet valve during backwash *)
        OUTLET_VALVE := FALSE;

        (* Activate backwash valve *)
        BACKWASH_VALVE := TRUE;

        (* Run backwash cycle *)
        BackwashTimer(IN := TRUE, PT := T#5M);
        IF BackwashTimer.Q THEN
            BACKWASH_VALVE := FALSE;
            FilterBackwashNeeded := FALSE;
            BackwashTimer(IN := FALSE);
            (* Restart filter operation timer *)
            FilterOperationTimer(IN := TRUE, PT := T#8H);
        END_IF
    END_IF

    (* UV System Control - final disinfection *)
    IF OUTLET_VALVE AND ScaledFlowRate > 20.0 THEN
        (* Activate UV when discharging *)
        UV_SYSTEM_START := TRUE;
    ELSE
        (* Turn off UV when not discharging to save energy *)
        UV_SYSTEM_START := FALSE;
    END_IF

END_IF

END_PROGRAM
